FUNCTION_BLOCK FB_WarehouseStock
VAR_INPUT	
END_VAR
VAR_OUTPUT
END_VAR
VAR
	iXAxis:				INT;
	iYAxis:				INT;
	bStored:			BOOL;
	bRemoved:			BOOL;
	arrStockPosition:	ARRAY[1..7, 1..12] OF INT;
	rMaxVal: 			REAL;
	rMinVal:			REAL;
	rMedVal:			REAL;
	rSum:				REAL;
END_VAR

METHOD M_Remove: 		BOOL
VAR_INPUT
	iProdNumber: 		INT;
END_VAR
bRemoved := FALSE;

IF iProdNumber = 0 THEN
	RETURN;
END_IF

FOR iXAxis := 1 TO 7 BY 1 DO
	FOR iYAxis :=  1 TO 12 BY 1 DO
		IF arrStockPosition[iXAxis, iYAxis] = iProdNumber THEN
			arrStockPosition[iXAxis, iYAxis] := 0;
			bRemoved := TRUE;
			EXIT;
		END_IF
		IF bRemoved = TRUE THEN
			RETURN;
		END_IF
	END_FOR
END_FOR
END_METHOD

METHOD M_Stats : BOOL
VAR_INPUT
END_VAR
FOR iXAxis := 1 TO 7 BY 1 DO
	FOR iYAxis :=  1 TO 12 BY 1 DO
		IF arrStockPosition[iXAxis, iYAxis] > 0 OR arrStockPosition[iXAxis, iYAxis] > rMaxVal THEN
			rMaxVal := arrStockPosition[iXAxis, iYAxis];
		END_IF
		IF arrStockPosition[iXAxis, iYAxis] < 3.402823E+38 OR arrStockPosition[iXAxis, iYAxis] < rMinVal THEN
			rMaxVal := arrStockPosition[iXAxis, iYAxis];
		END_IF
		rSum := 0 + arrStockPosition[iXAxis, iYAxis];
	END_FOR
END_FOR
rMedVal := rMedVal / (7*12);
END_METHOD

METHOD M_Store: 		BOOL
VAR_INPUT
	iProdNumber: 		INT;
END_VAR
bStored := FALSE;

IF iProdNumber = 0 THEN
	RETURN;
END_IF

FOR iXAxis := 1 TO 7 BY 1 DO
	FOR iYAxis :=  1 TO 12 BY 1 DO
		IF arrStockPosition[iXAxis, iYAxis] = 0 THEN
			arrStockPosition[iXAxis, iYAxis] := iProdNumber;
			bStored := TRUE;
			EXIT;
		END_IF
	END_FOR
	IF bStored = TRUE THEN
		RETURN;
		END_IF
END_FOR
END_METHOD

END_FUNCTION_BLOCK

(* stored: Version 1.1.0.1
   POU FB_WarehouseStock: Id {56887546-03b8-4afb-80a3-121d889fc915}, SpecialFunc None
   Method M_Remove: Id {0b9093b9-5d80-4a28-b602-596c4f7fc0e5}
   Method M_Stats: Id {8e8ac229-7d41-4b35-9101-a43ce4d54c3b}
   Method M_Store: Id {e43b1871-eb52-4cea-be35-e1eae7e91536} *)
